FUNCTION_BLOCK MOTOR_SWITCH (* Composite Function Block Type *)
  (* Standard: 61499-2 *)
  (* Version 0.0, 1/16/2023, Dmitrii, Flexbridge AB, template *)
  PACKAGE Main;
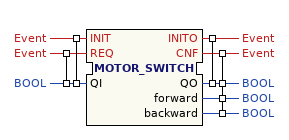
  EVENT_INPUT
    INIT WITH QI; (* Initialization Request *)
    REQ WITH QI; (* Normal Execution Request *)
  END_EVENT
  EVENT_OUTPUT
    INITO WITH QO; (* Initialization Confirm *)
    CNF WITH QO, forward, backward; (* Execution Confirmation *)
  END_EVENT
  VAR_INPUT
    QI : BOOL; (* Input event qualifier *)
  END_VAR
  VAR_OUTPUT
    QO : BOOL; (* Output event qualifier *)
    forward : BOOL;
    backward : BOOL;
  END_VAR
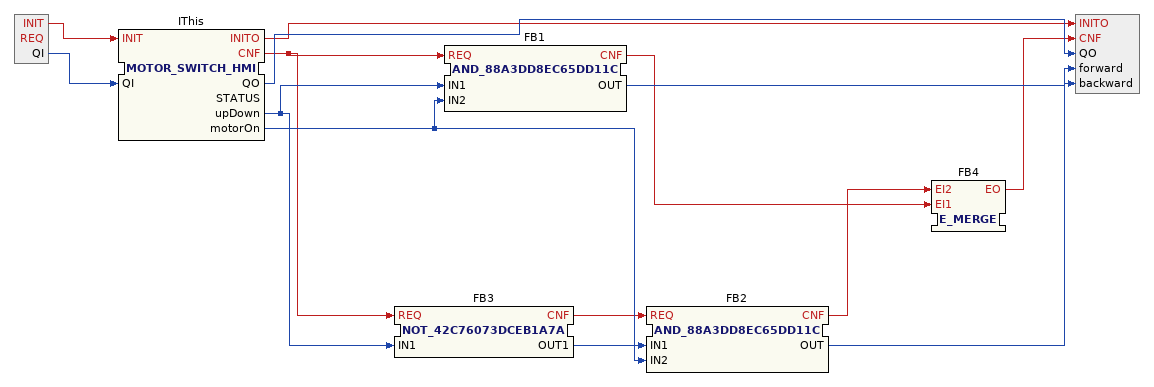
  FBS
    IThis : MOTOR_SWITCH_HMI;
    FB1 : AND_88A3DD8EC65DD11C; {SET_ATTRIBUTE(Configuration.GenericFBType.InterfaceParams, Runtime.Standard#CNT:=2;OUT:BOOL)}
    FB2 : AND_88A3DD8EC65DD11C; {SET_ATTRIBUTE(Configuration.GenericFBType.InterfaceParams, Runtime.Standard#CNT:=2;OUT:BOOL)}
    FB3 : NOT_42C76073DCEB1A7A; {SET_ATTRIBUTE(Configuration.GenericFBType.InterfaceParams, Runtime.Standard#CNT:=1;OUT${CNT$}:BOOL)}
    FB4 : E_MERGE;
  END_FBS
  EVENT_CONNECTIONS
    INIT TO IThis.INIT;
    IThis.CNF TO FB1.REQ;
    FB3.CNF TO FB2.REQ;
    IThis.CNF TO FB3.REQ;
    FB2.CNF TO FB4.EI2;
    FB1.CNF TO FB4.EI1;
    FB4.EO TO CNF;
    IThis.INITO TO INITO;
  END_CONNECTIONS
  DATA_CONNECTIONS
    QI TO IThis.QI;
    IThis.upDown TO FB1.IN1;
    IThis.motorOn TO FB1.IN2;
    FB1.OUT TO forward;
    FB3.OUT1 TO FB2.IN1;
    IThis.motorOn TO FB2.IN2;
    IThis.upDown TO FB3.IN1;
    FB2.OUT TO backward;
    IThis.QO TO QO;
  END_CONNECTIONS
END_FUNCTION_BLOCK
